PROGRAM MAIN
VAR	
END_VAR

TrafficLight(); // calling the function

END_PROGRAM

(* stored: Version 1.1.0.1, ProductVersion 3.1.4024.12
   POU MAIN: Id {d7b94376-8469-4017-9d71-930b5cb4c393}, SpecialFunc None *)
